// Mitsubishi GX Works2 project: 412_Coating_Code   PLC: Q03UDE

PROGRAM MAIN
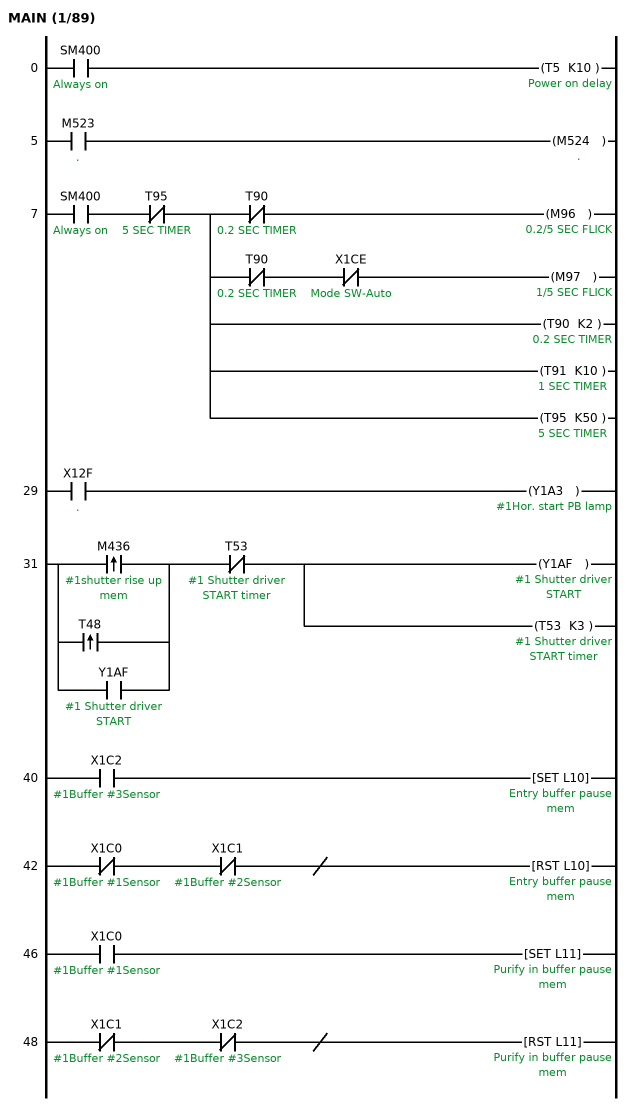
0     LD      SM400  ; Always on
      OUT     T5 K10  ; Power on delay
5     LD      M523  ; .
      OUT     M524  ; .
7     LD      SM400  ; Always on
      ANI     T95  ; 5 SEC TIMER
      MPS
      ANI     T90  ; 0.2 SEC TIMER
      OUT     M96  ; 0.2/5 SEC FLICK
      MRD
      ANI     T90  ; 0.2 SEC TIMER
      ANI     X1CE  ; Mode SW-Auto
      OUT     M97  ; 1/5 SEC FLICK
      MPP
      OUT     T90 K2  ; 0.2 SEC TIMER
      OUT     T91 K10  ; 1 SEC TIMER
      OUT     T95 K50  ; 5 SEC TIMER
29    LD      X12F  ; .
      OUT     Y1A3  ; #1Hor. start PB lamp
31    LDP     M436  ; #1shutter rise up mem
      ORP     T48
      OR      Y1AF  ; #1 Shutter driver START
      ANI     T53  ; #1 Shutter driver START timer
      OUT     Y1AF  ; #1 Shutter driver START
      OUT     T53 K3  ; #1 Shutter driver START timer
40    LD      X1C2  ; #1Buffer #3Sensor
      SET     L10  ; Entry buffer pause mem
42    LDI     X1C0  ; #1Buffer #1Sensor
      ANI     X1C1  ; #1Buffer #2Sensor
      INV
      RST     L10  ; Entry buffer pause mem
46    LD      X1C0  ; #1Buffer #1Sensor
      SET     L11  ; Purify in buffer pause mem
48    LDI     X1C1  ; #1Buffer #2Sensor
      ANI     X1C2  ; #1Buffer #3Sensor
      INV
      RST     L11  ; Purify in buffer pause mem
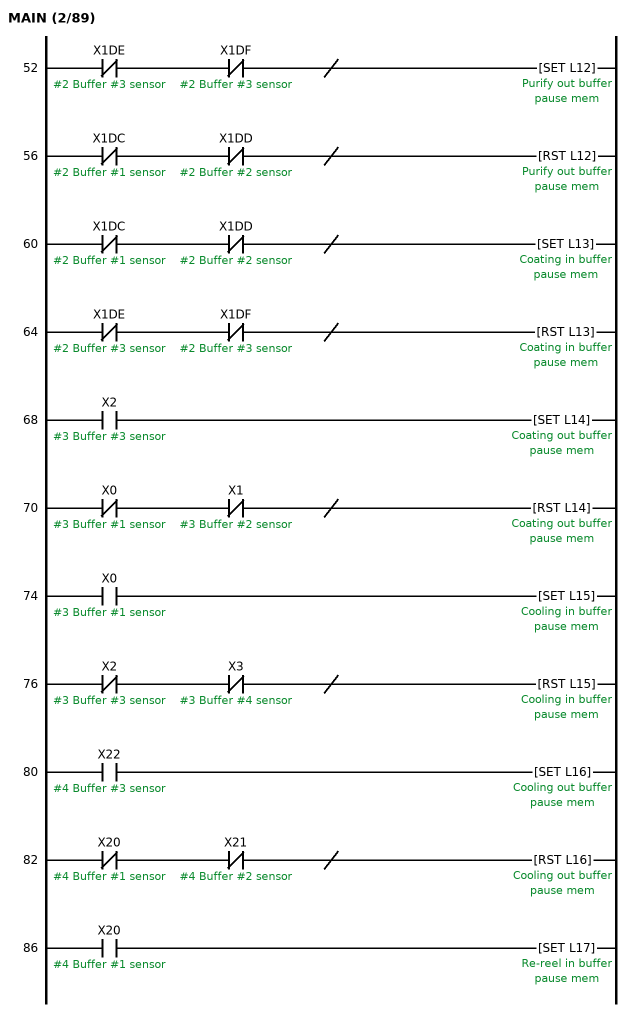
52    LDI     X1DE  ; #2 Buffer #3 sensor
      ANI     X1DF  ; #2 Buffer #3 sensor
      INV
      SET     L12  ; Purify out buffer pause mem
56    LDI     X1DC  ; #2 Buffer #1 sensor
      ANI     X1DD  ; #2 Buffer #2 sensor
      INV
      RST     L12  ; Purify out buffer pause mem
60    LDI     X1DC  ; #2 Buffer #1 sensor
      ANI     X1DD  ; #2 Buffer #2 sensor
      INV
      SET     L13  ; Coating in buffer pause mem
64    LDI     X1DE  ; #2 Buffer #3 sensor
      ANI     X1DF  ; #2 Buffer #3 sensor
      INV
      RST     L13  ; Coating in buffer pause mem
68    LD      X2  ; #3 Buffer #3 sensor
      SET     L14  ; Coating out buffer pause mem
70    LDI     X0  ; #3 Buffer #1 sensor
      ANI     X1  ; #3 Buffer #2 sensor
      INV
      RST     L14  ; Coating out buffer pause mem
74    LD      X0  ; #3 Buffer #1 sensor
      SET     L15  ; Cooling in buffer pause mem
76    LDI     X2  ; #3 Buffer #3 sensor
      ANI     X3  ; #3 Buffer #4 sensor
      INV
      RST     L15  ; Cooling in buffer pause mem
80    LD      X22  ; #4 Buffer #3 sensor
      SET     L16  ; Cooling out buffer pause mem
82    LDI     X20  ; #4 Buffer #1 sensor
      ANI     X21  ; #4 Buffer #2 sensor
      INV
      RST     L16  ; Cooling out buffer pause mem
86    LD      X20  ; #4 Buffer #1 sensor
      SET     L17  ; Re-reel in buffer pause mem
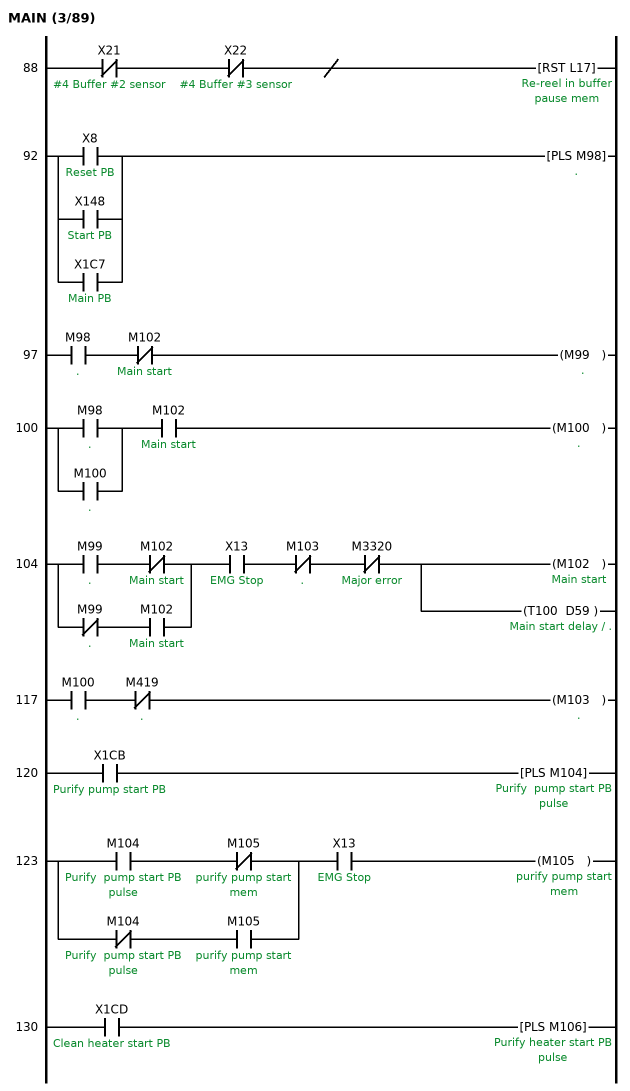
88    LDI     X21  ; #4 Buffer #2 sensor
      ANI     X22  ; #4 Buffer #3 sensor
      INV
      RST     L17  ; Re-reel in buffer pause mem
92    LD      X8  ; Reset PB
      OR      X148  ; Start PB
      OR      X1C7  ; Main PB
      PLS     M98  ; .
97    LD      M98  ; .
      ANI     M102  ; Main start
      OUT     M99  ; .
100   LD      M98  ; .
      OR      M100  ; .
      AND     M102  ; Main start
      OUT     M100  ; .
104   LD      M99  ; .
      ANI     M102  ; Main start
      LDI     M99  ; .
      AND     M102  ; Main start
      ORB
      AND     X13  ; EMG Stop
      ANI     M103  ; .
      ANI     M3320  ; Major error
      OUT     M102  ; Main start
      OUT     T100 D59  ; Main start delay / .
117   LD      M100  ; .
      ANI     M419  ; .
      OUT     M103  ; .
120   LD      X1CB  ; Purify pump start PB
      PLS     M104  ; Purify  pump start PB pulse
123   LD      M104  ; Purify  pump start PB pulse
      ANI     M105  ; purify pump start mem
      LDI     M104  ; Purify  pump start PB pulse
      AND     M105  ; purify pump start mem
      ORB
      AND     X13  ; EMG Stop
      OUT     M105  ; purify pump start mem
130   LD      X1CD  ; Clean heater start PB
      PLS     M106  ; Purify heater start PB pulse
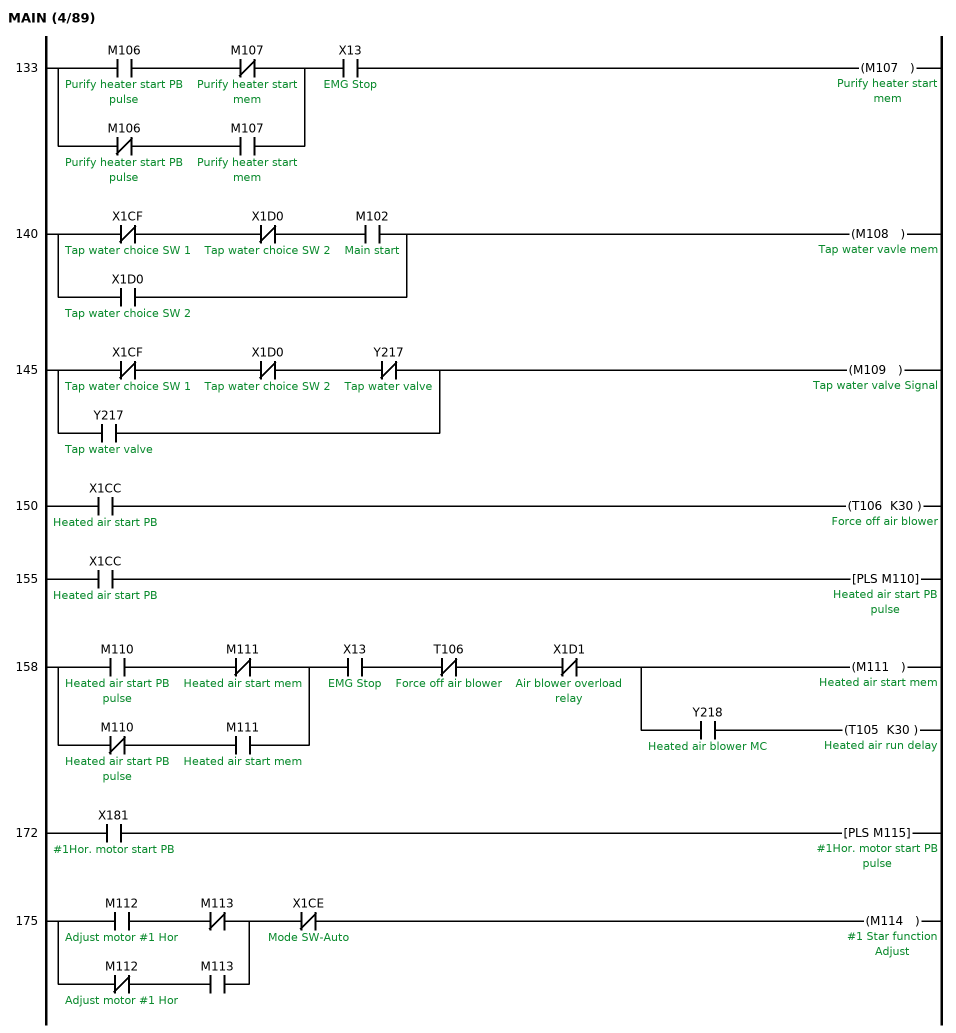
133   LD      M106  ; Purify heater start PB pulse
      ANI     M107  ; Purify heater start mem
      LDI     M106  ; Purify heater start PB pulse
      AND     M107  ; Purify heater start mem
      ORB
      AND     X13  ; EMG Stop
      OUT     M107  ; Purify heater start mem
140   LDI     X1CF  ; Tap water choice SW 1
      ANI     X1D0  ; Tap water choice SW 2
      AND     M102  ; Main start
      OR      X1D0  ; Tap water choice SW 2
      OUT     M108  ; Tap water vavle mem
145   LDI     X1CF  ; Tap water choice SW 1
      ANI     X1D0  ; Tap water choice SW 2
      ANI     Y217  ; Tap water valve
      OR      Y217  ; Tap water valve
      OUT     M109  ; Tap water valve Signal
150   LD      X1CC  ; Heated air start PB
      OUT     T106 K30  ; Force off air blower
155   LD      X1CC  ; Heated air start PB
      PLS     M110  ; Heated air start PB pulse
158   LD      M110  ; Heated air start PB pulse
      ANI     M111  ; Heated air start mem
      LDI     M110  ; Heated air start PB pulse
      AND     M111  ; Heated air start mem
      ORB
      AND     X13  ; EMG Stop
      ANI     T106  ; Force off air blower
      ANI     X1D1  ; Air blower overload relay
      OUT     M111  ; Heated air start mem
      AND     Y218  ; Heated air blower MC
      OUT     T105 K30  ; Heated air run delay
172   LD      X181  ; #1Hor. motor start PB
      PLS     M115  ; #1Hor. motor start PB pulse
175   LD      M112  ; Adjust motor #1 Hor
      ANI     M113
      LDI     M112  ; Adjust motor #1 Hor
      AND     M113
      ORB
      ANI     X1CE  ; Mode SW-Auto
      OUT     M114  ; #1 Star function Adjust
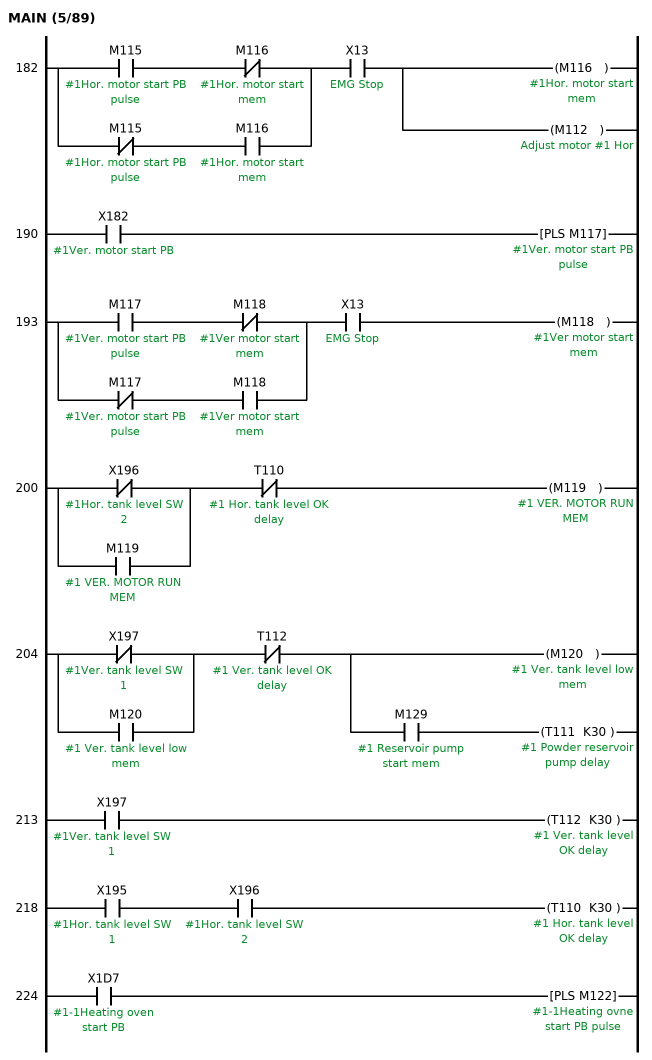
182   LD      M115  ; #1Hor. motor start PB pulse
      ANI     M116  ; #1Hor. motor start mem
      LDI     M115  ; #1Hor. motor start PB pulse
      AND     M116  ; #1Hor. motor start mem
      ORB
      AND     X13  ; EMG Stop
      OUT     M116  ; #1Hor. motor start mem
      OUT     M112  ; Adjust motor #1 Hor
190   LD      X182  ; #1Ver. motor start PB
      PLS     M117  ; #1Ver. motor start PB pulse
193   LD      M117  ; #1Ver. motor start PB pulse
      ANI     M118  ; #1Ver motor start mem
      LDI     M117  ; #1Ver. motor start PB pulse
      AND     M118  ; #1Ver motor start mem
      ORB
      AND     X13  ; EMG Stop
      OUT     M118  ; #1Ver motor start mem
200   LDI     X196  ; #1Hor. tank level SW 2
      OR      M119  ; #1 VER. MOTOR RUN MEM
      ANI     T110  ; #1 Hor. tank level OK delay
      OUT     M119  ; #1 VER. MOTOR RUN MEM
204   LDI     X197  ; #1Ver. tank level SW 1
      OR      M120  ; #1 Ver. tank level low mem
      ANI     T112  ; #1 Ver. tank level OK delay
      OUT     M120  ; #1 Ver. tank level low mem
      AND     M129  ; #1 Reservoir pump start mem
      OUT     T111 K30  ; #1 Powder reservoir pump delay
213   LD      X197  ; #1Ver. tank level SW 1
      OUT     T112 K30  ; #1 Ver. tank level OK delay
218   LD      X195  ; #1Hor. tank level SW 1
      AND     X196  ; #1Hor. tank level SW 2
      OUT     T110 K30  ; #1 Hor. tank level OK delay
224   LD      X1D7  ; #1-1Heating oven start PB
      PLS     M122  ; #1-1Heating ovne start PB pulse
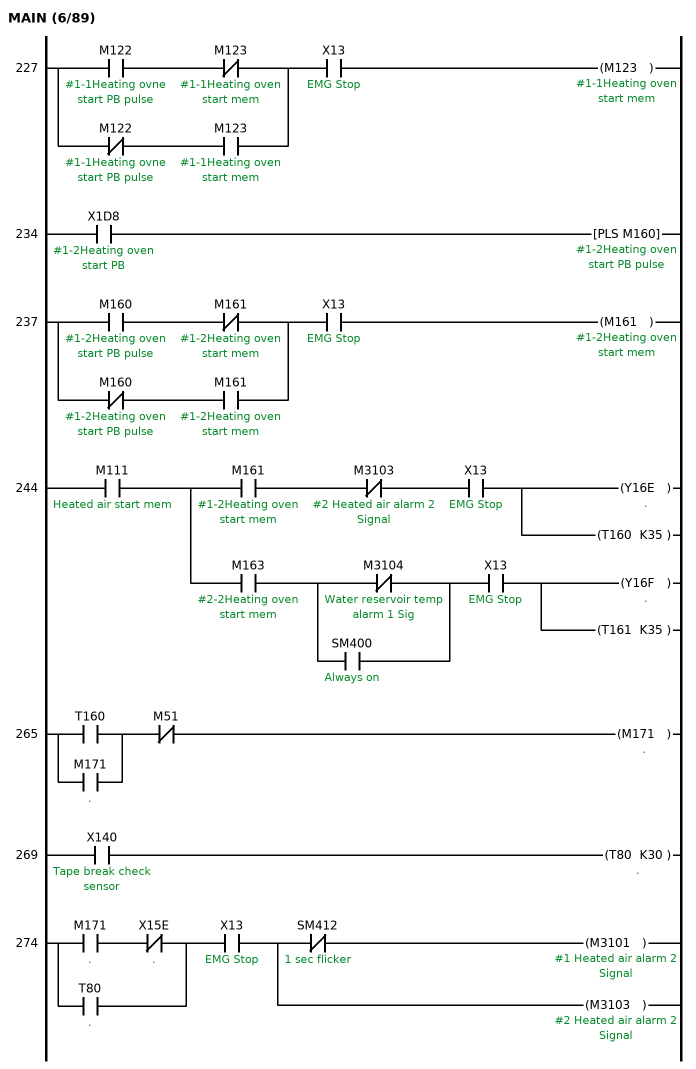
227   LD      M122  ; #1-1Heating ovne start PB pulse
      ANI     M123  ; #1-1Heating oven start mem
      LDI     M122  ; #1-1Heating ovne start PB pulse
      AND     M123  ; #1-1Heating oven start mem
      ORB
      AND     X13  ; EMG Stop
      OUT     M123  ; #1-1Heating oven start mem
234   LD      X1D8  ; #1-2Heating oven start PB
      PLS     M160  ; #1-2Heating oven start PB pulse
237   LD      M160  ; #1-2Heating oven start PB pulse
      ANI     M161  ; #1-2Heating oven start mem
      LDI     M160  ; #1-2Heating oven start PB pulse
      AND     M161  ; #1-2Heating oven start mem
      ORB
      AND     X13  ; EMG Stop
      OUT     M161  ; #1-2Heating oven start mem
244   LD      M111  ; Heated air start mem
      MPS
      AND     M161  ; #1-2Heating oven start mem
      ANI     M3103  ; #2 Heated air alarm 2 Signal
      AND     X13  ; EMG Stop
      OUT     Y16E  ; .
      OUT     T160 K35
      MPP
      AND     M163  ; #2-2Heating oven start mem
      LDI     M3104  ; Water reservoir temp alarm 1 Sig
      OR      SM400  ; Always on
      ANB
      AND     X13  ; EMG Stop
      OUT     Y16F  ; .
      OUT     T161 K35
265   LD      T160
      OR      M171  ; .
      ANI     M51
      OUT     M171  ; .
269   LD      X140  ; Tape break check sensor
      OUT     T80 K30  ; .
274   LD      M171  ; .
      ANI     X15E  ; .
      OR      T80  ; .
      AND     X13  ; EMG Stop
      MPS
      ANI     SM412  ; 1 sec flicker
      OUT     M3101  ; #1 Heated air alarm 2 Signal
      MPP
      OUT     M3103  ; #2 Heated air alarm 2 Signal
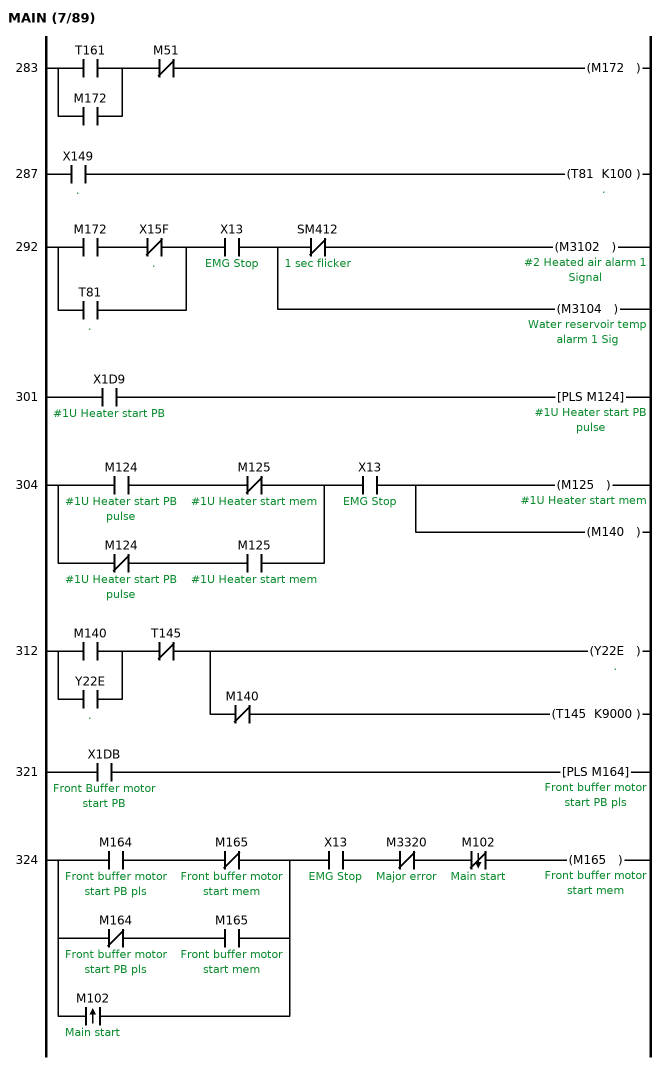
283   LD      T161
      OR      M172
      ANI     M51
      OUT     M172
287   LD      X149  ; .
      OUT     T81 K100  ; .
292   LD      M172
      ANI     X15F  ; .
      OR      T81  ; .
      AND     X13  ; EMG Stop
      MPS
      ANI     SM412  ; 1 sec flicker
      OUT     M3102  ; #2 Heated air alarm 1 Signal
      MPP
      OUT     M3104  ; Water reservoir temp alarm 1 Sig
301   LD      X1D9  ; #1U Heater start PB
      PLS     M124  ; #1U Heater start PB pulse
304   LD      M124  ; #1U Heater start PB pulse
      ANI     M125  ; #1U Heater start mem
      LDI     M124  ; #1U Heater start PB pulse
      AND     M125  ; #1U Heater start mem
      ORB
      AND     X13  ; EMG Stop
      OUT     M125  ; #1U Heater start mem
      OUT     M140
312   LD      M140
      OR      Y22E  ; .
      ANI     T145
      OUT     Y22E  ; .
      ANI     M140
      OUT     T145 K9000
321   LD      X1DB  ; Front Buffer motor start PB
      PLS     M164  ; Front buffer motor start PB pls
324   LD      M164  ; Front buffer motor start PB pls
      ANI     M165  ; Front buffer motor start mem
      LDI     M164  ; Front buffer motor start PB pls
      AND     M165  ; Front buffer motor start mem
      ORB
      ORP     M102  ; Main start
      AND     X13  ; EMG Stop
      ANI     M3320  ; Major error
      ANDFI   M102  ; Main start
      OUT     M165  ; Front buffer motor start mem
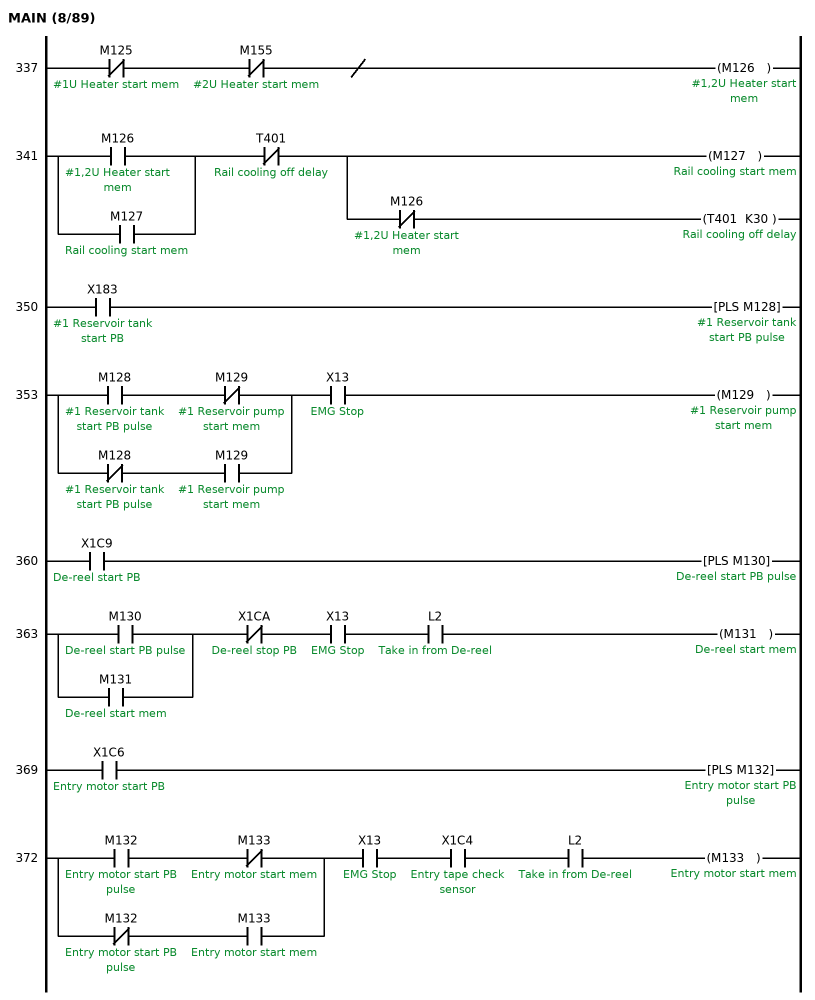
337   LDI     M125  ; #1U Heater start mem
      ANI     M155  ; #2U Heater start mem
      INV
      OUT     M126  ; #1,2U Heater start mem
341   LD      M126  ; #1,2U Heater start mem
      OR      M127  ; Rail cooling start mem
      ANI     T401  ; Rail cooling off delay
      OUT     M127  ; Rail cooling start mem
      ANI     M126  ; #1,2U Heater start mem
      OUT     T401 K30  ; Rail cooling off delay
350   LD      X183  ; #1 Reservoir tank start PB
      PLS     M128  ; #1 Reservoir tank start PB pulse
353   LD      M128  ; #1 Reservoir tank start PB pulse
      ANI     M129  ; #1 Reservoir pump start mem
      LDI     M128  ; #1 Reservoir tank start PB pulse
      AND     M129  ; #1 Reservoir pump start mem
      ORB
      AND     X13  ; EMG Stop
      OUT     M129  ; #1 Reservoir pump start mem
360   LD      X1C9  ; De-reel start PB
      PLS     M130  ; De-reel start PB pulse
363   LD      M130  ; De-reel start PB pulse
      OR      M131  ; De-reel start mem
      ANI     X1CA  ; De-reel stop PB
      AND     X13  ; EMG Stop
      AND     L2  ; Take in from De-reel
      OUT     M131  ; De-reel start mem
369   LD      X1C6  ; Entry motor start PB
      PLS     M132  ; Entry motor start PB pulse
372   LD      M132  ; Entry motor start PB pulse
      ANI     M133  ; Entry motor start mem
      LDI     M132  ; Entry motor start PB pulse
      AND     M133  ; Entry motor start mem
      ORB
      AND     X13  ; EMG Stop
      AND     X1C4  ; Entry tape check sensor
      AND     L2  ; Take in from De-reel
      OUT     M133  ; Entry motor start mem
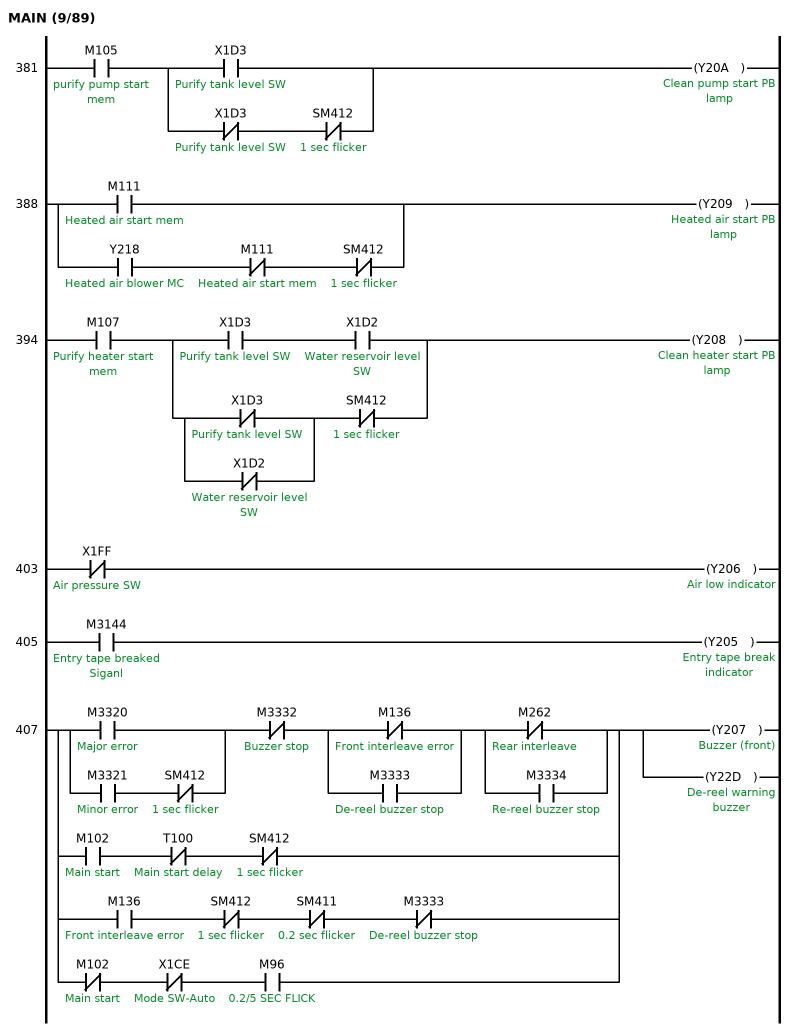
381   LD      M105  ; purify pump start mem
      LD      X1D3  ; Purify tank level SW
      LDI     X1D3  ; Purify tank level SW
      ANI     SM412  ; 1 sec flicker
      ORB
      ANB
      OUT     Y20A  ; Clean pump start PB lamp
388   LD      M111  ; Heated air start mem
      LD      Y218  ; Heated air blower MC
      ANI     M111  ; Heated air start mem
      ANI     SM412  ; 1 sec flicker
      ORB
      OUT     Y209  ; Heated air start PB lamp
394   LD      M107  ; Purify heater start mem
      LD      X1D3  ; Purify tank level SW
      AND     X1D2  ; Water reservoir level SW
      LDI     X1D3  ; Purify tank level SW
      ORI     X1D2  ; Water reservoir level SW
      ANI     SM412  ; 1 sec flicker
      ORB
      ANB
      OUT     Y208  ; Clean heater start PB lamp
403   LDI     X1FF  ; Air pressure SW
      OUT     Y206  ; Air low indicator
405   LD      M3144  ; Entry tape breaked Siganl
      OUT     Y205  ; Entry tape break indicator
407   LD      M3320  ; Major error
      LD      M3321  ; Minor error
      ANI     SM412  ; 1 sec flicker
      ORB
      ANI     M3332  ; Buzzer stop
      LDI     M136  ; Front interleave error
      OR      M3333  ; De-reel buzzer stop
      ANB
      LDI     M262  ; Rear interleave
      OR      M3334  ; Re-reel buzzer stop
      ANB
      LD      M102  ; Main start
      ANI     T100  ; Main start delay
      ANI     SM412  ; 1 sec flicker
      ORB
      LD      M136  ; Front interleave error
      ANI     SM412  ; 1 sec flicker
      ANI     SM411  ; 0.2 sec flicker
      ANI     M3333  ; De-reel buzzer stop
      ORB
      LDI     M102  ; Main start
      ANI     X1CE  ; Mode SW-Auto
      AND     M96  ; 0.2/5 SEC FLICK
      ORB
      OUT     Y207  ; Buzzer (front)
      OUT     Y22D  ; De-reel warning buzzer
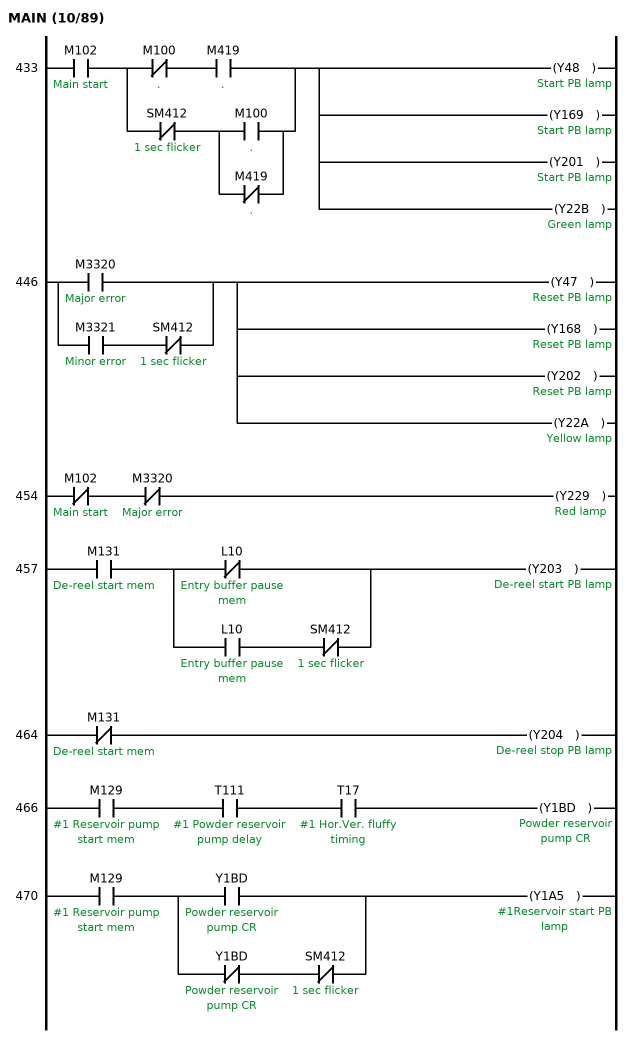
433   LD      M102  ; Main start
      LDI     M100  ; .
      AND     M419  ; .
      LDI     SM412  ; 1 sec flicker
      LD      M100  ; .
      ORI     M419  ; .
      ANB
      ORB
      ANB
      OUT     Y48  ; Start PB lamp
      OUT     Y169  ; Start PB lamp
      OUT     Y201  ; Start PB lamp
      OUT     Y22B  ; Green lamp
446   LD      M3320  ; Major error
      LD      M3321  ; Minor error
      ANI     SM412  ; 1 sec flicker
      ORB
      OUT     Y47  ; Reset PB lamp
      OUT     Y168  ; Reset PB lamp
      OUT     Y202  ; Reset PB lamp
      OUT     Y22A  ; Yellow lamp
454   LDI     M102  ; Main start
      ANI     M3320  ; Major error
      OUT     Y229  ; Red lamp
457   LD      M131  ; De-reel start mem
      LDI     L10  ; Entry buffer pause mem
      LD      L10  ; Entry buffer pause mem
      ANI     SM412  ; 1 sec flicker
      ORB
      ANB
      OUT     Y203  ; De-reel start PB lamp
464   LDI     M131  ; De-reel start mem
      OUT     Y204  ; De-reel stop PB lamp
466   LD      M129  ; #1 Reservoir pump start mem
      AND     T111  ; #1 Powder reservoir pump delay
      AND     T17  ; #1 Hor.Ver. fluffy timing
      OUT     Y1BD  ; Powder reservoir pump CR
470   LD      M129  ; #1 Reservoir pump start mem
      LD      Y1BD  ; Powder reservoir pump CR
      LDI     Y1BD  ; Powder reservoir pump CR
      ANI     SM412  ; 1 sec flicker
      ORB
      ANB
      OUT     Y1A5  ; #1Reservoir start PB lamp
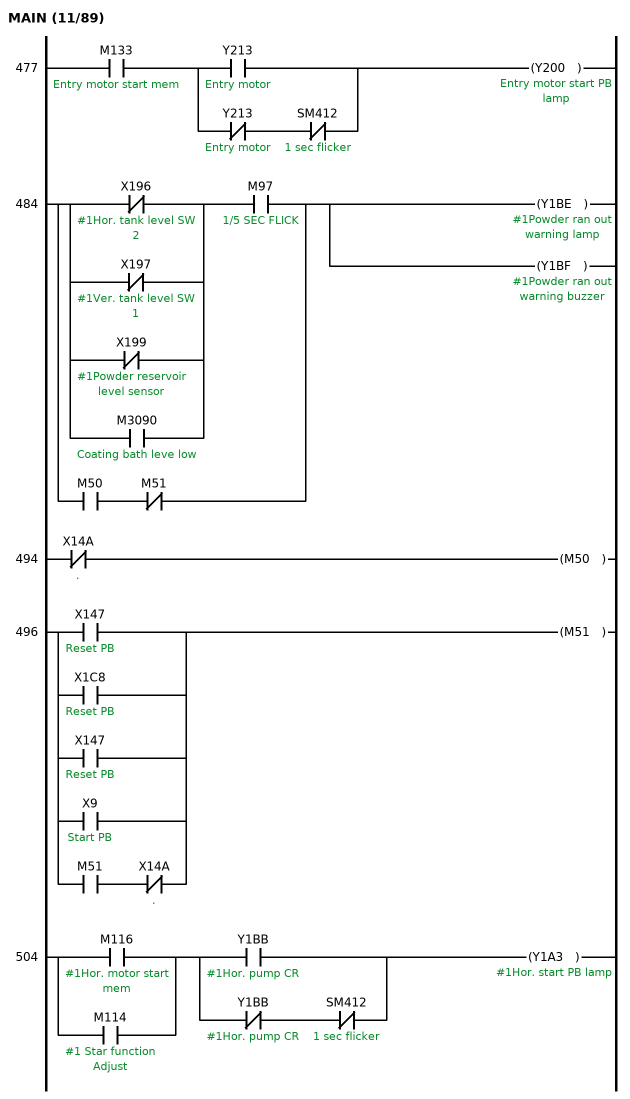
477   LD      M133  ; Entry motor start mem
      LD      Y213  ; Entry motor
      LDI     Y213  ; Entry motor
      ANI     SM412  ; 1 sec flicker
      ORB
      ANB
      OUT     Y200  ; Entry motor start PB lamp
484   LDI     X196  ; #1Hor. tank level SW 2
      ORI     X197  ; #1Ver. tank level SW 1
      ORI     X199  ; #1Powder reservoir level sensor
      OR      M3090  ; Coating bath leve low
      AND     M97  ; 1/5 SEC FLICK
      LD      M50
      ANI     M51
      ORB
      OUT     Y1BE  ; #1Powder ran out warning lamp
      OUT     Y1BF  ; #1Powder ran out warning buzzer
494   LDI     X14A  ; .
      OUT     M50
496   LD      X147  ; Reset PB
      OR      X1C8  ; Reset PB
      OR      X147  ; Reset PB
      OR      X9  ; Start PB
      LD      M51
      ANI     X14A  ; .
      ORB
      OUT     M51
504   LD      M116  ; #1Hor. motor start mem
      OR      M114  ; #1 Star function Adjust
      LD      Y1BB  ; #1Hor. pump CR
      LDI     Y1BB  ; #1Hor. pump CR
      ANI     SM412  ; 1 sec flicker
      ORB
      ANB
      OUT     Y1A3  ; #1Hor. start PB lamp
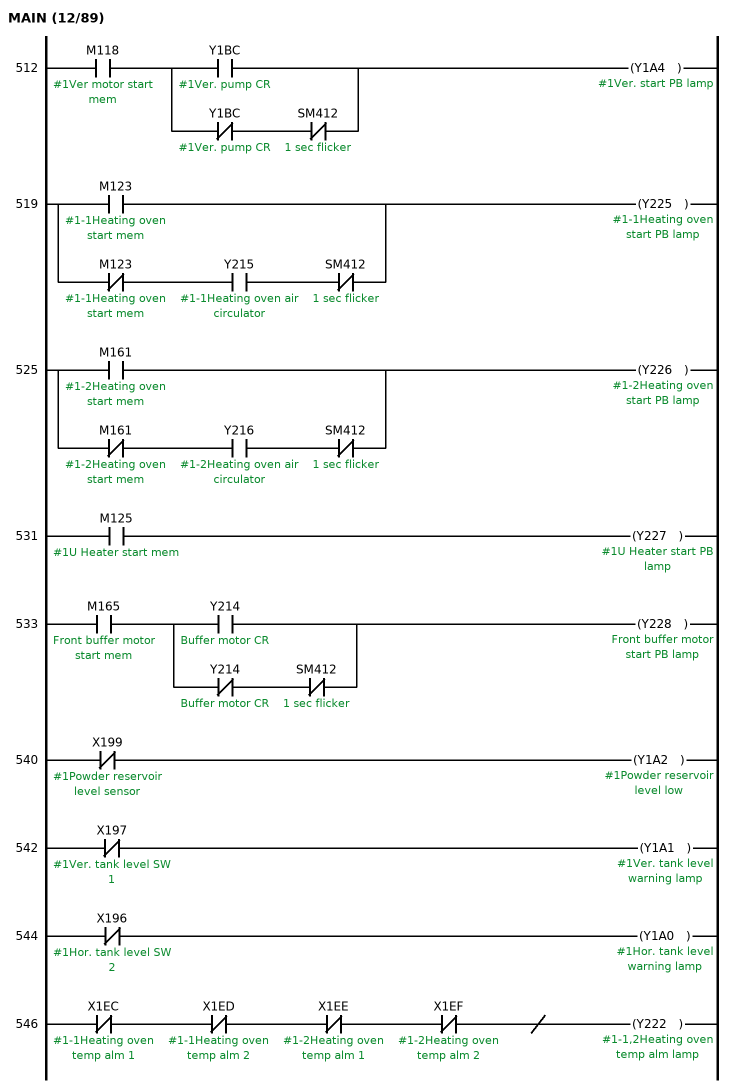
512   LD      M118  ; #1Ver motor start mem
      LD      Y1BC  ; #1Ver. pump CR
      LDI     Y1BC  ; #1Ver. pump CR
      ANI     SM412  ; 1 sec flicker
      ORB
      ANB
      OUT     Y1A4  ; #1Ver. start PB lamp
519   LD      M123  ; #1-1Heating oven start mem
      LDI     M123  ; #1-1Heating oven start mem
      AND     Y215  ; #1-1Heating oven air circulator
      ANI     SM412  ; 1 sec flicker
      ORB
      OUT     Y225  ; #1-1Heating oven start PB lamp
525   LD      M161  ; #1-2Heating oven start mem
      LDI     M161  ; #1-2Heating oven start mem
      AND     Y216  ; #1-2Heating oven air circulator
      ANI     SM412  ; 1 sec flicker
      ORB
      OUT     Y226  ; #1-2Heating oven start PB lamp
531   LD      M125  ; #1U Heater start mem
      OUT     Y227  ; #1U Heater start PB lamp
533   LD      M165  ; Front buffer motor start mem
      LD      Y214  ; Buffer motor CR
      LDI     Y214  ; Buffer motor CR
      ANI     SM412  ; 1 sec flicker
      ORB
      ANB
      OUT     Y228  ; Front buffer motor start PB lamp
540   LDI     X199  ; #1Powder reservoir level sensor
      OUT     Y1A2  ; #1Powder reservoir level low
542   LDI     X197  ; #1Ver. tank level SW 1
      OUT     Y1A1  ; #1Ver. tank level warning lamp
544   LDI     X196  ; #1Hor. tank level SW 2
      OUT     Y1A0  ; #1Hor. tank level warning lamp
546   LDI     X1EC  ; #1-1Heating oven temp alm 1
      ANI     X1ED  ; #1-1Heating oven temp alm 2
      ANI     X1EE  ; #1-2Heating oven temp alm 1
      ANI     X1EF  ; #1-2Heating oven temp alm 2
      INV
      OUT     Y222  ; #1-1,2Heating oven temp alm lamp
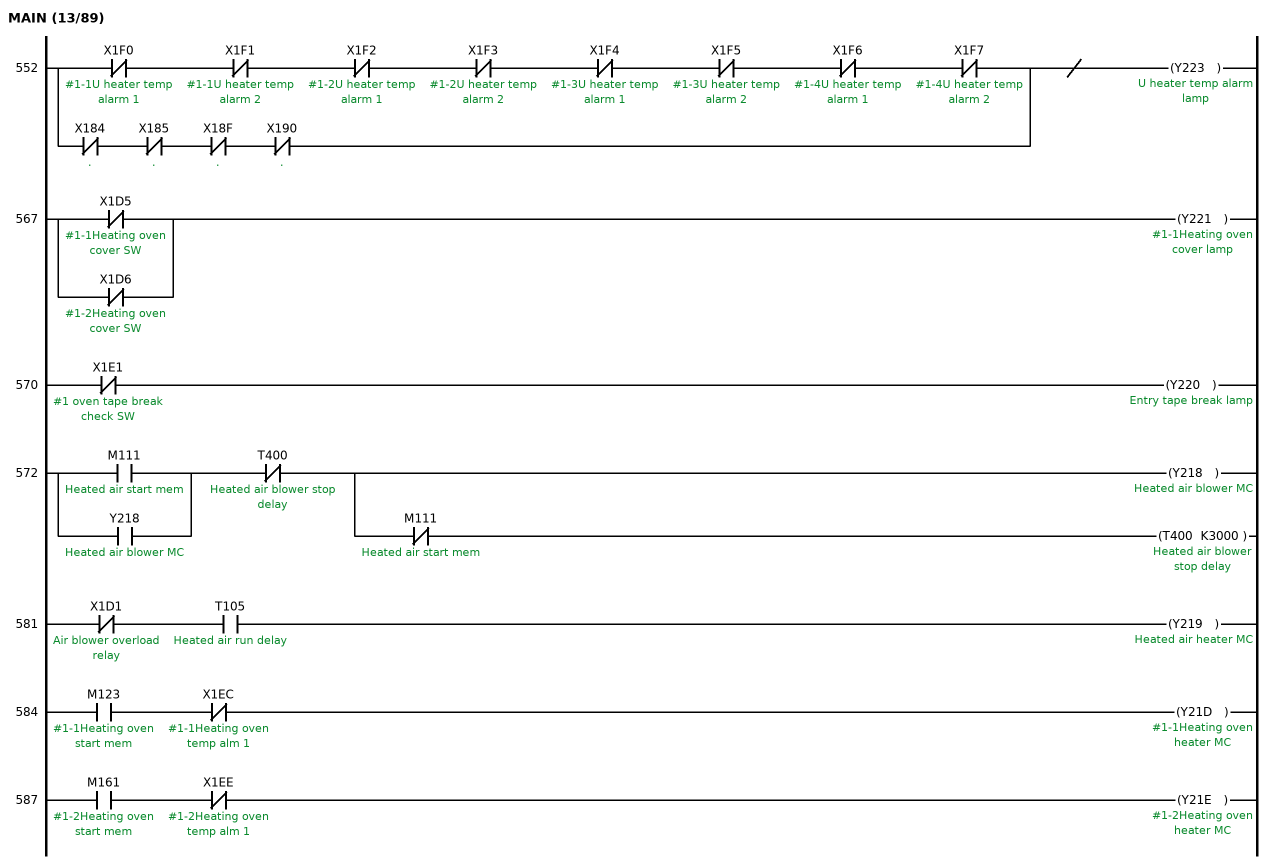
552   LDI     X1F0  ; #1-1U heater temp alarm 1
      ANI     X1F1  ; #1-1U heater temp alarm 2
      ANI     X1F2  ; #1-2U heater temp alarm 1
      ANI     X1F3  ; #1-2U heater temp alarm 2
      ANI     X1F4  ; #1-3U heater temp alarm 1
      ANI     X1F5  ; #1-3U heater temp alarm 2
      ANI     X1F6  ; #1-4U heater temp alarm 1
      ANI     X1F7  ; #1-4U heater temp alarm 2
      LDI     X184  ; .
      ANI     X185  ; .
      ANI     X18F  ; .
      ANI     X190  ; .
      ORB
      INV
      OUT     Y223  ; U heater temp alarm lamp
567   LDI     X1D5  ; #1-1Heating oven cover SW
      ORI     X1D6  ; #1-2Heating oven cover SW
      OUT     Y221  ; #1-1Heating oven cover lamp
570   LDI     X1E1  ; #1 oven tape break check SW
      OUT     Y220  ; Entry tape break lamp
572   LD      M111  ; Heated air start mem
      OR      Y218  ; Heated air blower MC
      ANI     T400  ; Heated air blower stop delay
      OUT     Y218  ; Heated air blower MC
      ANI     M111  ; Heated air start mem
      OUT     T400 K3000  ; Heated air blower stop delay
581   LDI     X1D1  ; Air blower overload relay
      AND     T105  ; Heated air run delay
      OUT     Y219  ; Heated air heater MC
584   LD      M123  ; #1-1Heating oven start mem
      ANI     X1EC  ; #1-1Heating oven temp alm 1
      OUT     Y21D  ; #1-1Heating oven heater MC
587   LD      M161  ; #1-2Heating oven start mem
      ANI     X1EE  ; #1-2Heating oven temp alm 1
      OUT     Y21E  ; #1-2Heating oven heater MC
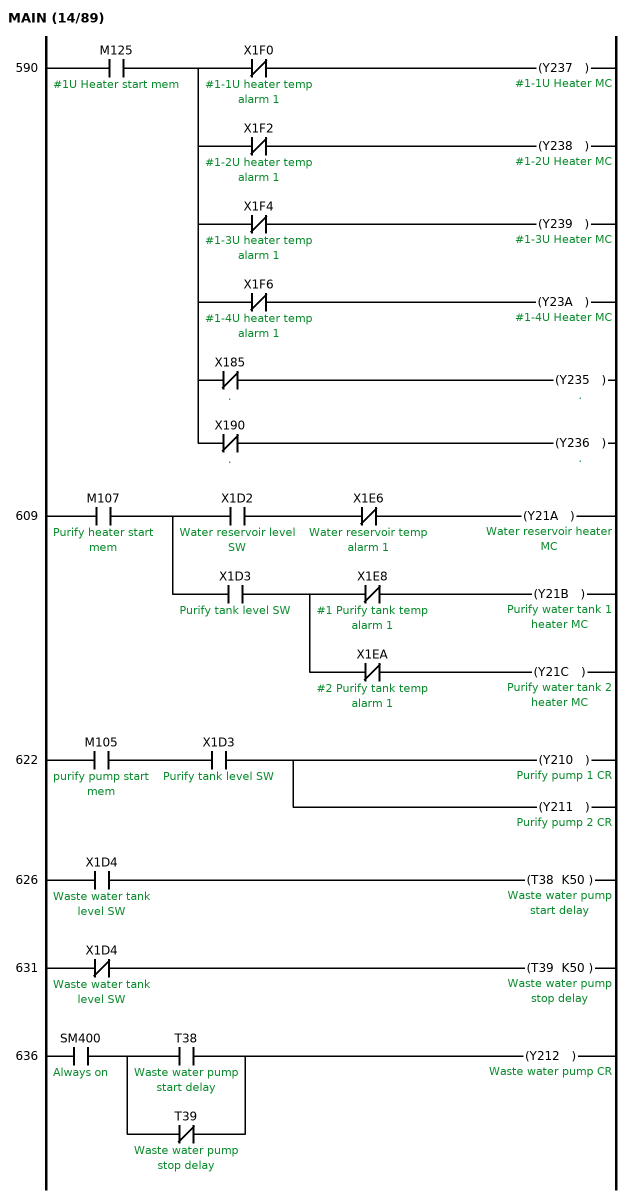
590   LD      M125  ; #1U Heater start mem
      MPS
      ANI     X1F0  ; #1-1U heater temp alarm 1
      OUT     Y237  ; #1-1U Heater MC
      MRD
      ANI     X1F2  ; #1-2U heater temp alarm 1
      OUT     Y238  ; #1-2U Heater MC
      MRD
      ANI     X1F4  ; #1-3U heater temp alarm 1
      OUT     Y239  ; #1-3U Heater MC
      MRD
      ANI     X1F6  ; #1-4U heater temp alarm 1
      OUT     Y23A  ; #1-4U Heater MC
      MRD
      ANI     X185  ; .
      OUT     Y235  ; .
      MPP
      ANI     X190  ; .
      OUT     Y236  ; .
609   LD      M107  ; Purify heater start mem
      MPS
      AND     X1D2  ; Water reservoir level SW
      ANI     X1E6  ; Water reservoir temp alarm 1
      OUT     Y21A  ; Water reservoir heater MC
      MPP
      AND     X1D3  ; Purify tank level SW
      MPS
      ANI     X1E8  ; #1 Purify tank temp alarm 1
      OUT     Y21B  ; Purify water tank 1 heater MC
      MPP
      ANI     X1EA  ; #2 Purify tank temp alarm 1
      OUT     Y21C  ; Purify water tank 2 heater MC
622   LD      M105  ; purify pump start mem
      AND     X1D3  ; Purify tank level SW
      OUT     Y210  ; Purify pump 1 CR
      OUT     Y211  ; Purify pump 2 CR
626   LD      X1D4  ; Waste water tank level SW
      OUT     T38 K50  ; Waste water pump start delay
631   LDI     X1D4  ; Waste water tank level SW
      OUT     T39 K50  ; Waste water pump stop delay
636   LD      SM400  ; Always on
      LD      T38  ; Waste water pump start delay
      ORI     T39  ; Waste water pump stop delay
      ANB
      OUT     Y212  ; Waste water pump CR
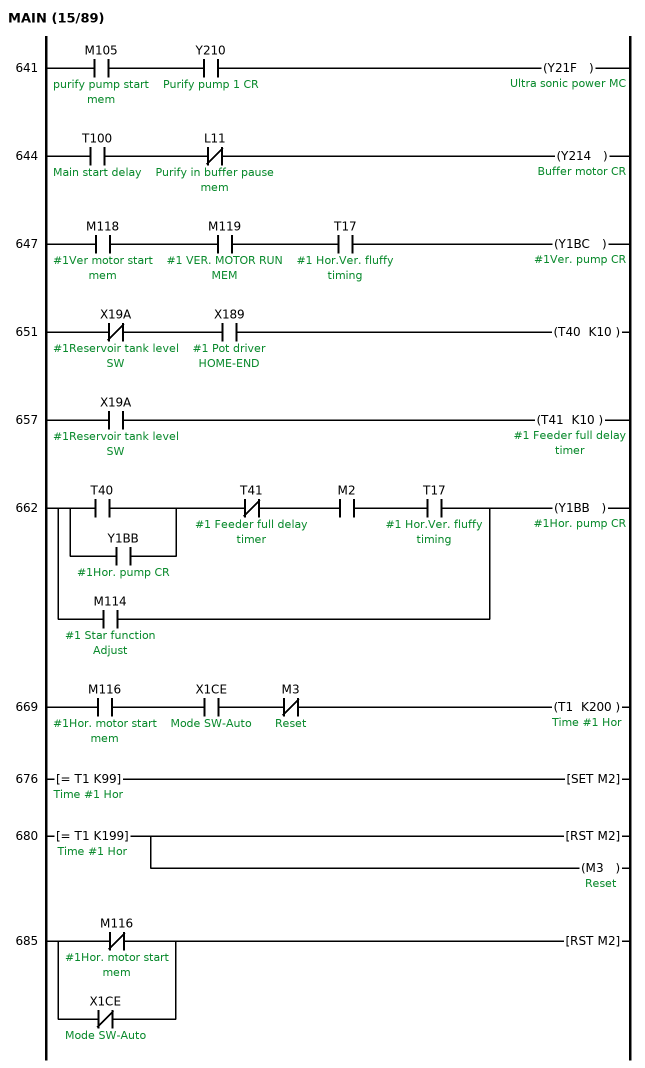
641   LD      M105  ; purify pump start mem
      AND     Y210  ; Purify pump 1 CR
      OUT     Y21F  ; Ultra sonic power MC
644   LD      T100  ; Main start delay
      ANI     L11  ; Purify in buffer pause mem
      OUT     Y214  ; Buffer motor CR
647   LD      M118  ; #1Ver motor start mem
      AND     M119  ; #1 VER. MOTOR RUN MEM
      AND     T17  ; #1 Hor.Ver. fluffy timing
      OUT     Y1BC  ; #1Ver. pump CR
651   LDI     X19A  ; #1Reservoir tank level SW
      AND     X189  ; #1 Pot driver HOME-END
      OUT     T40 K10
657   LD      X19A  ; #1Reservoir tank level SW
      OUT     T41 K10  ; #1 Feeder full delay timer
662   LD      T40
      OR      Y1BB  ; #1Hor. pump CR
      ANI     T41  ; #1 Feeder full delay timer
      AND     M2
      AND     T17  ; #1 Hor.Ver. fluffy timing
      OR      M114  ; #1 Star function Adjust
      OUT     Y1BB  ; #1Hor. pump CR
669   LD      M116  ; #1Hor. motor start mem
      AND     X1CE  ; Mode SW-Auto
      ANI     M3  ; Reset
      OUT     T1 K200  ; Time #1 Hor
676   LD=     T1 K99  ; Time #1 Hor
      SET     M2
680   LD=     T1 K199  ; Time #1 Hor
      RST     M2
      OUT     M3  ; Reset
685   LDI     M116  ; #1Hor. motor start mem
      ORI     X1CE  ; Mode SW-Auto
      RST     M2
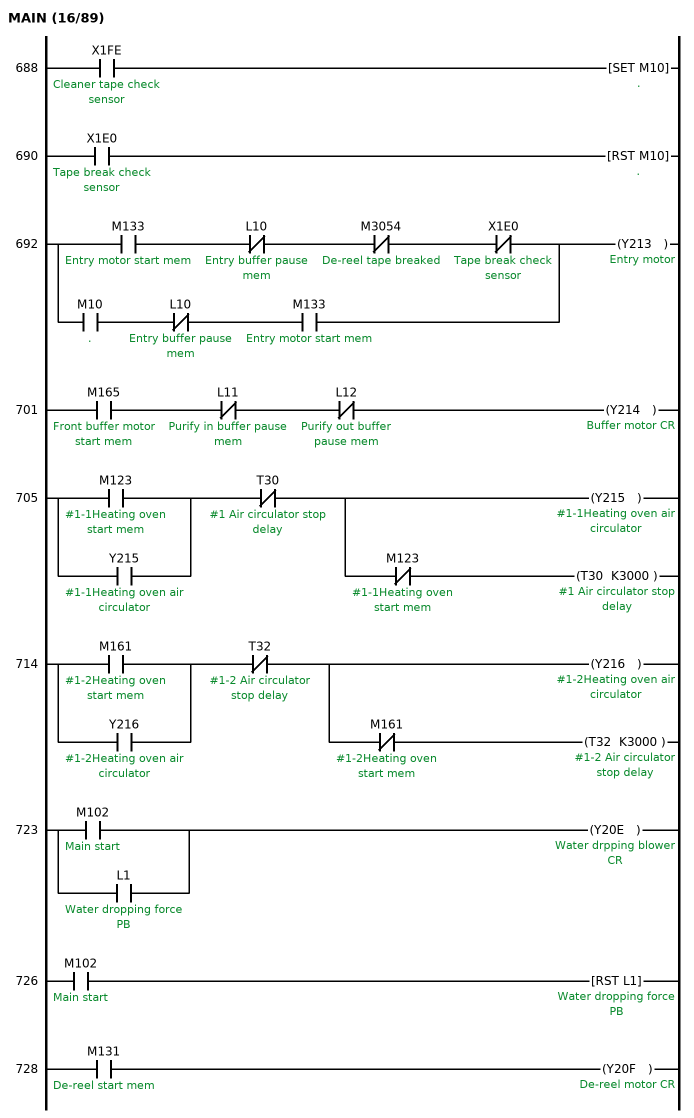
688   LD      X1FE  ; Cleaner tape check sensor
      SET     M10  ; .
690   LD      X1E0  ; Tape break check sensor
      RST     M10  ; .
692   LD      M133  ; Entry motor start mem
      ANI     L10  ; Entry buffer pause mem
      ANI     M3054  ; De-reel tape breaked
      ANI     X1E0  ; Tape break check sensor
      LD      M10  ; .
      ANI     L10  ; Entry buffer pause mem
      AND     M133  ; Entry motor start mem
      ORB
      OUT     Y213  ; Entry motor
701   LD      M165  ; Front buffer motor start mem
      ANI     L11  ; Purify in buffer pause mem
      ANI     L12  ; Purify out buffer pause mem
      OUT     Y214  ; Buffer motor CR
705   LD      M123  ; #1-1Heating oven start mem
      OR      Y215  ; #1-1Heating oven air circulator
      ANI     T30  ; #1 Air circulator stop delay
      OUT     Y215  ; #1-1Heating oven air circulator
      ANI     M123  ; #1-1Heating oven start mem
      OUT     T30 K3000  ; #1 Air circulator stop delay
714   LD      M161  ; #1-2Heating oven start mem
      OR      Y216  ; #1-2Heating oven air circulator
      ANI     T32  ; #1-2 Air circulator stop delay
      OUT     Y216  ; #1-2Heating oven air circulator
      ANI     M161  ; #1-2Heating oven start mem
      OUT     T32 K3000  ; #1-2 Air circulator stop delay
723   LD      M102  ; Main start
      OR      L1  ; Water dropping force PB
      OUT     Y20E  ; Water drpping blower CR
726   LD      M102  ; Main start
      RST     L1  ; Water dropping force PB
728   LD      M131  ; De-reel start mem
      OUT     Y20F  ; De-reel motor CR
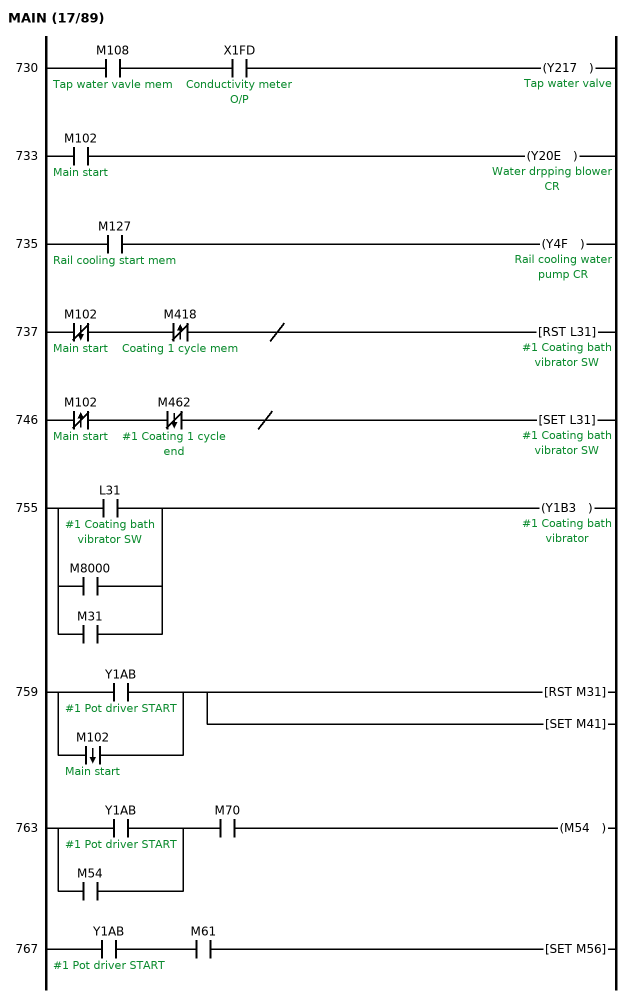
730   LD      M108  ; Tap water vavle mem
      AND     X1FD  ; Conductivity meter O/P
      OUT     Y217  ; Tap water valve
733   LD      M102  ; Main start
      OUT     Y20E  ; Water drpping blower CR
735   LD      M127  ; Rail cooling start mem
      OUT     Y4F  ; Rail cooling water pump CR
737   LDFI    M102  ; Main start
      ANDPI   M418  ; Coating 1 cycle mem
      INV
      RST     L31  ; #1 Coating bath vibrator SW
746   LDPI    M102  ; Main start
      ANDFI   M462  ; #1 Coating 1 cycle end
      INV
      SET     L31  ; #1 Coating bath vibrator SW
755   LD      L31  ; #1 Coating bath vibrator SW
      OR      M8000
      OR      M31
      OUT     Y1B3  ; #1 Coating bath vibrator
759   LD      Y1AB  ; #1 Pot driver START
      ORF     M102  ; Main start
      RST     M31
      SET     M41
763   LD      Y1AB  ; #1 Pot driver START
      OR      M54
      AND     M70
      OUT     M54
767   LD      Y1AB  ; #1 Pot driver START
      AND     M61
      SET     M56
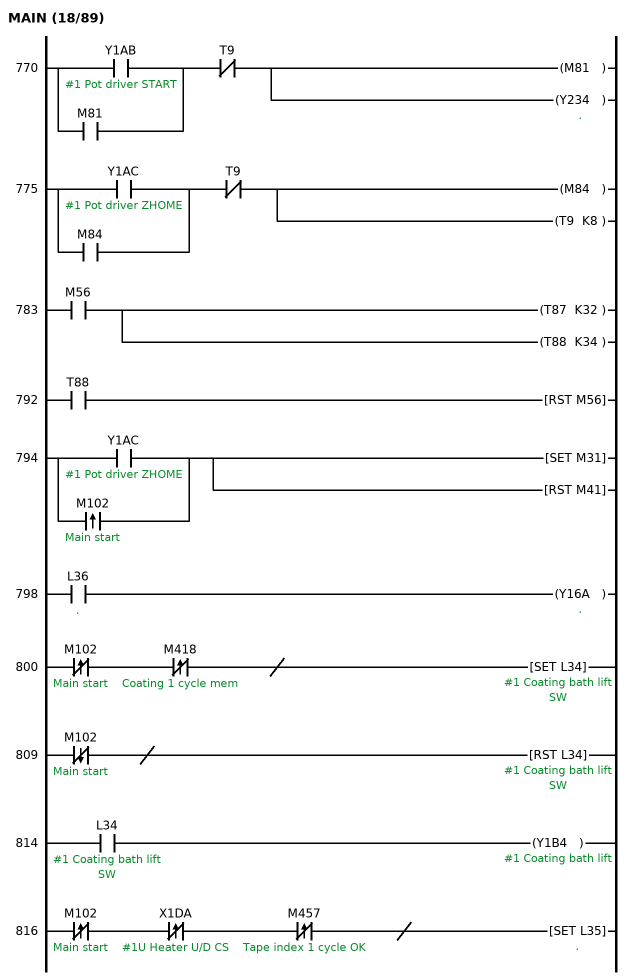
770   LD      Y1AB  ; #1 Pot driver START
      OR      M81
      ANI     T9
      OUT     M81
      OUT     Y234  ; .
775   LD      Y1AC  ; #1 Pot driver ZHOME
      OR      M84
      ANI     T9
      OUT     M84
      OUT     T9 K8
783   LD      M56
      OUT     T87 K32
      OUT     T88 K34
792   LD      T88
      RST     M56
794   LD      Y1AC  ; #1 Pot driver ZHOME
      ORP     M102  ; Main start
      SET     M31
      RST     M41
798   LD      L36  ; .
      OUT     Y16A  ; .
800   LDPI    M102  ; Main start
      ANDPI   M418  ; Coating 1 cycle mem
      INV
      SET     L34  ; #1 Coating bath lift SW
809   LDFI    M102  ; Main start
      INV
      RST     L34  ; #1 Coating bath lift SW
814   LD      L34  ; #1 Coating bath lift SW
      OUT     Y1B4  ; #1 Coating bath lift
816   LDPI    M102  ; Main start
      ANDPI   X1DA  ; #1U Heater U/D CS
      ANDPI   M457  ; Tape index 1 cycle OK
      INV
      SET     L35  ; .
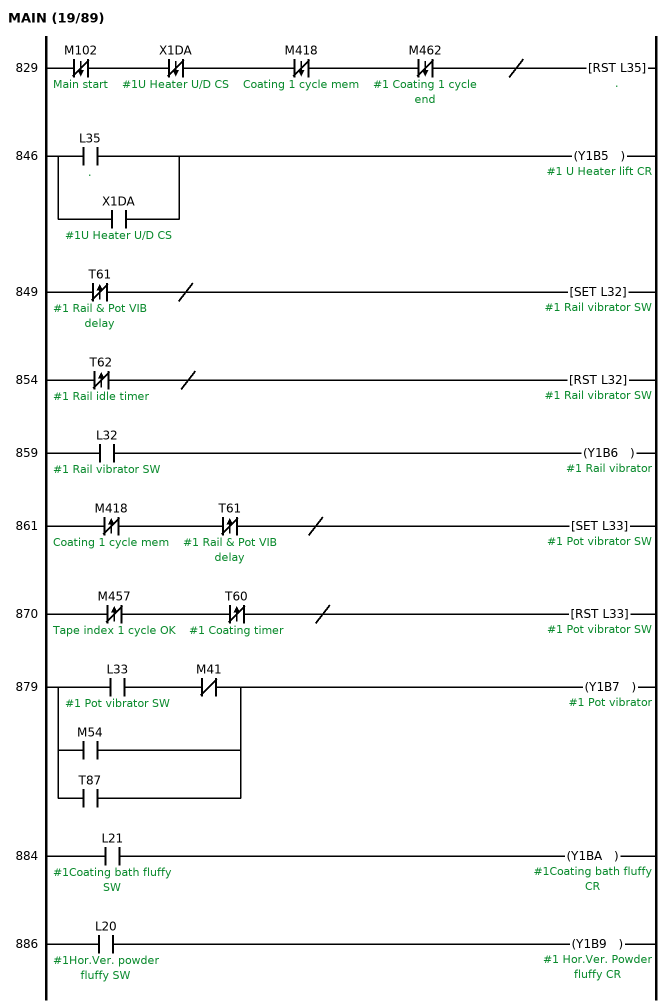
829   LDFI    M102  ; Main start
      ANDFI   X1DA  ; #1U Heater U/D CS
      ANDFI   M418  ; Coating 1 cycle mem
      ANDFI   M462  ; #1 Coating 1 cycle end
      INV
      RST     L35  ; .
846   LD      L35  ; .
      OR      X1DA  ; #1U Heater U/D CS
      OUT     Y1B5  ; #1 U Heater lift CR
849   LDPI    T61  ; #1 Rail & Pot VIB delay
      INV
      SET     L32  ; #1 Rail vibrator SW
854   LDPI    T62  ; #1 Rail idle timer
      INV
      RST     L32  ; #1 Rail vibrator SW
859   LD      L32  ; #1 Rail vibrator SW
      OUT     Y1B6  ; #1 Rail vibrator
861   LDPI    M418  ; Coating 1 cycle mem
      ANDPI   T61  ; #1 Rail & Pot VIB delay
      INV
      SET     L33  ; #1 Pot vibrator SW
870   LDPI    M457  ; Tape index 1 cycle OK
      ANDPI   T60  ; #1 Coating timer
      INV
      RST     L33  ; #1 Pot vibrator SW
879   LD      L33  ; #1 Pot vibrator SW
      ANI     M41
      OR      M54
      OR      T87
      OUT     Y1B7  ; #1 Pot vibrator
884   LD      L21  ; #1Coating bath fluffy SW
      OUT     Y1BA  ; #1Coating bath fluffy CR
886   LD      L20  ; #1Hor.Ver. powder fluffy SW
      OUT     Y1B9  ; #1 Hor.Ver. Powder fluffy CR
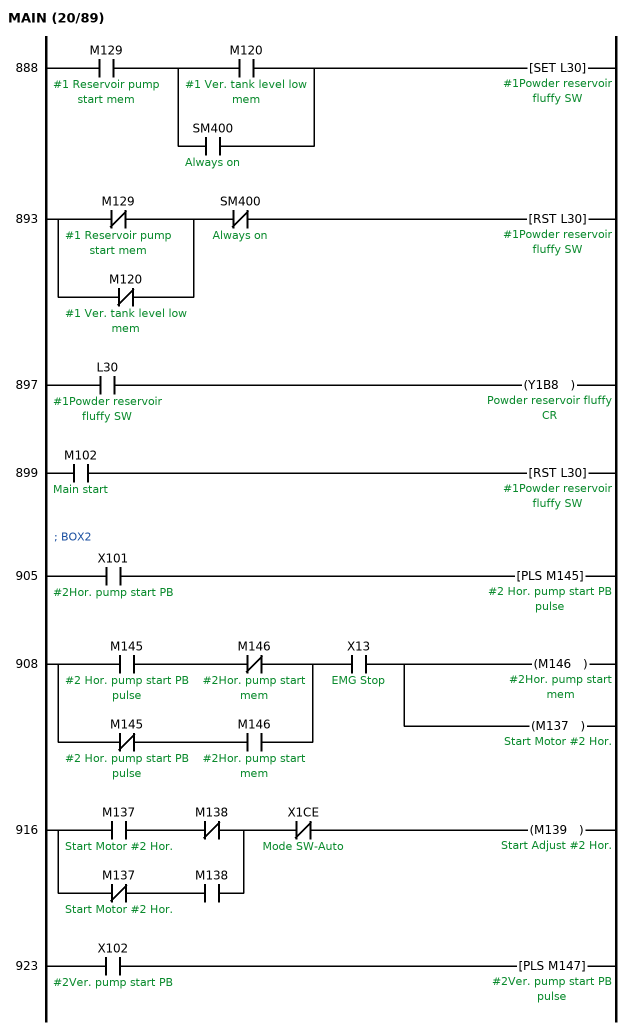
888   LD      M129  ; #1 Reservoir pump start mem
      LD      M120  ; #1 Ver. tank level low mem
      OR      SM400  ; Always on
      ANB
      SET     L30  ; #1Powder reservoir fluffy SW
893   LDI     M129  ; #1 Reservoir pump start mem
      ORI     M120  ; #1 Ver. tank level low mem
      ANI     SM400  ; Always on
      RST     L30  ; #1Powder reservoir fluffy SW
897   LD      L30  ; #1Powder reservoir fluffy SW
      OUT     Y1B8  ; Powder reservoir fluffy CR
899   LD      M102  ; Main start
      RST     L30  ; #1Powder reservoir fluffy SW
; BOX2
905   LD      X101  ; #2Hor. pump start PB
      PLS     M145  ; #2 Hor. pump start PB pulse
908   LD      M145  ; #2 Hor. pump start PB pulse
      ANI     M146  ; #2Hor. pump start mem
      LDI     M145  ; #2 Hor. pump start PB pulse
      AND     M146  ; #2Hor. pump start mem
      ORB
      AND     X13  ; EMG Stop
      OUT     M146  ; #2Hor. pump start mem
      OUT     M137  ; Start Motor #2 Hor.
916   LD      M137  ; Start Motor #2 Hor.
      ANI     M138
      LDI     M137  ; Start Motor #2 Hor.
      AND     M138
      ORB
      ANI     X1CE  ; Mode SW-Auto
      OUT     M139  ; Start Adjust #2 Hor.
923   LD      X102  ; #2Ver. pump start PB
      PLS     M147  ; #2Ver. pump start PB pulse
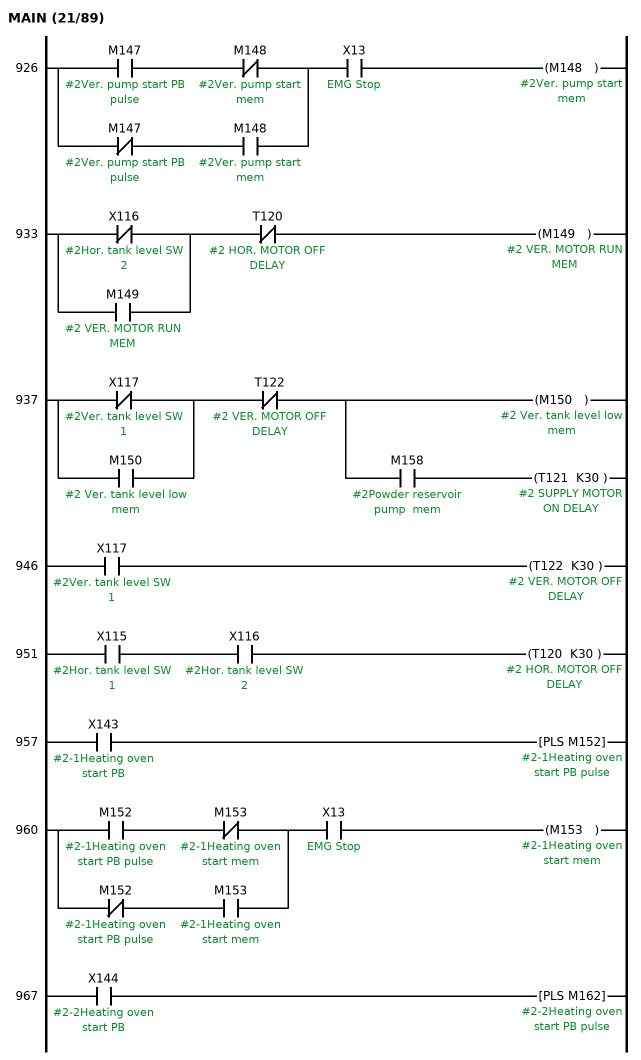
926   LD      M147  ; #2Ver. pump start PB pulse
      ANI     M148  ; #2Ver. pump start mem
      LDI     M147  ; #2Ver. pump start PB pulse
      AND     M148  ; #2Ver. pump start mem
      ORB
      AND     X13  ; EMG Stop
      OUT     M148  ; #2Ver. pump start mem
933   LDI     X116  ; #2Hor. tank level SW 2
      OR      M149  ; #2 VER. MOTOR RUN MEM
      ANI     T120  ; #2 HOR. MOTOR OFF DELAY
      OUT     M149  ; #2 VER. MOTOR RUN MEM
937   LDI     X117  ; #2Ver. tank level SW 1
      OR      M150  ; #2 Ver. tank level low mem
      ANI     T122  ; #2 VER. MOTOR OFF DELAY
      OUT     M150  ; #2 Ver. tank level low mem
      AND     M158  ; #2Powder reservoir pump  mem
      OUT     T121 K30  ; #2 SUPPLY MOTOR ON DELAY
946   LD      X117  ; #2Ver. tank level SW 1
      OUT     T122 K30  ; #2 VER. MOTOR OFF DELAY
951   LD      X115  ; #2Hor. tank level SW 1
      AND     X116  ; #2Hor. tank level SW 2
      OUT     T120 K30  ; #2 HOR. MOTOR OFF DELAY
957   LD      X143  ; #2-1Heating oven start PB
      PLS     M152  ; #2-1Heating oven start PB pulse
960   LD      M152  ; #2-1Heating oven start PB pulse
      ANI     M153  ; #2-1Heating oven start mem
      LDI     M152  ; #2-1Heating oven start PB pulse
      AND     M153  ; #2-1Heating oven start mem
      ORB
      AND     X13  ; EMG Stop
      OUT     M153  ; #2-1Heating oven start mem
967   LD      X144  ; #2-2Heating oven start PB
      PLS     M162  ; #2-2Heating oven start PB pulse
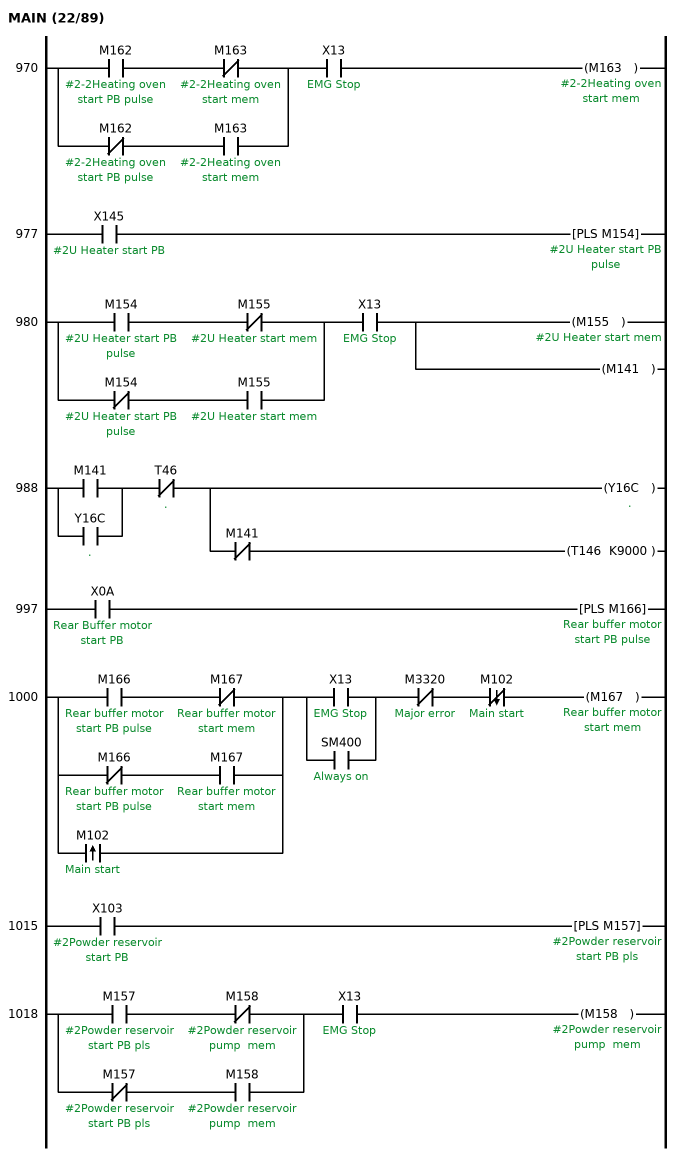
970   LD      M162  ; #2-2Heating oven start PB pulse
      ANI     M163  ; #2-2Heating oven start mem
      LDI     M162  ; #2-2Heating oven start PB pulse
      AND     M163  ; #2-2Heating oven start mem
      ORB
      AND     X13  ; EMG Stop
      OUT     M163  ; #2-2Heating oven start mem
977   LD      X145  ; #2U Heater start PB
      PLS     M154  ; #2U Heater start PB pulse
980   LD      M154  ; #2U Heater start PB pulse
      ANI     M155  ; #2U Heater start mem
      LDI     M154  ; #2U Heater start PB pulse
      AND     M155  ; #2U Heater start mem
      ORB
      AND     X13  ; EMG Stop
      OUT     M155  ; #2U Heater start mem
      OUT     M141
988   LD      M141
      OR      Y16C  ; .
      ANI     T46  ; .
      OUT     Y16C  ; .
      ANI     M141
      OUT     T146 K9000
997   LD      X0A  ; Rear Buffer motor start PB
      PLS     M166  ; Rear buffer motor start PB pulse
1000  LD      M166  ; Rear buffer motor start PB pulse
      ANI     M167  ; Rear buffer motor start mem
      LDI     M166  ; Rear buffer motor start PB pulse
      AND     M167  ; Rear buffer motor start mem
      ORB
      ORP     M102  ; Main start
      LD      X13  ; EMG Stop
      OR      SM400  ; Always on
      ANB
      ANI     M3320  ; Major error
      ANDFI   M102  ; Main start
      OUT     M167  ; Rear buffer motor start mem
1015  LD      X103  ; #2Powder reservoir start PB
      PLS     M157  ; #2Powder reservoir start PB pls
1018  LD      M157  ; #2Powder reservoir start PB pls
      ANI     M158  ; #2Powder reservoir pump  mem
      LDI     M157  ; #2Powder reservoir start PB pls
      AND     M158  ; #2Powder reservoir pump  mem
      ORB
      AND     X13  ; EMG Stop
      OUT     M158  ; #2Powder reservoir pump  mem
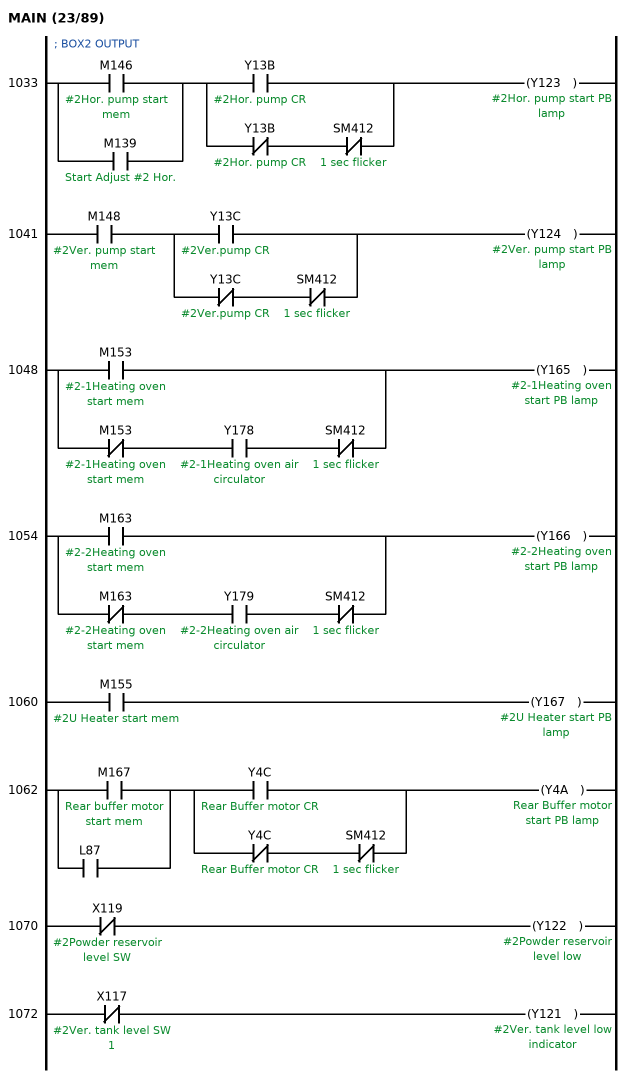
; BOX2 OUTPUT
1033  LD      M146  ; #2Hor. pump start mem
      OR      M139  ; Start Adjust #2 Hor.
      LD      Y13B  ; #2Hor. pump CR
      LDI     Y13B  ; #2Hor. pump CR
      ANI     SM412  ; 1 sec flicker
      ORB
      ANB
      OUT     Y123  ; #2Hor. pump start PB lamp
1041  LD      M148  ; #2Ver. pump start mem
      LD      Y13C  ; #2Ver.pump CR
      LDI     Y13C  ; #2Ver.pump CR
      ANI     SM412  ; 1 sec flicker
      ORB
      ANB
      OUT     Y124  ; #2Ver. pump start PB lamp
1048  LD      M153  ; #2-1Heating oven start mem
      LDI     M153  ; #2-1Heating oven start mem
      AND     Y178  ; #2-1Heating oven air circulator
      ANI     SM412  ; 1 sec flicker
      ORB
      OUT     Y165  ; #2-1Heating oven start PB lamp
1054  LD      M163  ; #2-2Heating oven start mem
      LDI     M163  ; #2-2Heating oven start mem
      AND     Y179  ; #2-2Heating oven air circulator
      ANI     SM412  ; 1 sec flicker
      ORB
      OUT     Y166  ; #2-2Heating oven start PB lamp
1060  LD      M155  ; #2U Heater start mem
      OUT     Y167  ; #2U Heater start PB lamp
1062  LD      M167  ; Rear buffer motor start mem
      OR      L87
      LD      Y4C  ; Rear Buffer motor CR
      LDI     Y4C  ; Rear Buffer motor CR
      ANI     SM412  ; 1 sec flicker
      ORB
      ANB
      OUT     Y4A  ; Rear Buffer motor start PB lamp
1070  LDI     X119  ; #2Powder reservoir level SW
      OUT     Y122  ; #2Powder reservoir level low
1072  LDI     X117  ; #2Ver. tank level SW 1
      OUT     Y121  ; #2Ver. tank level low indicator
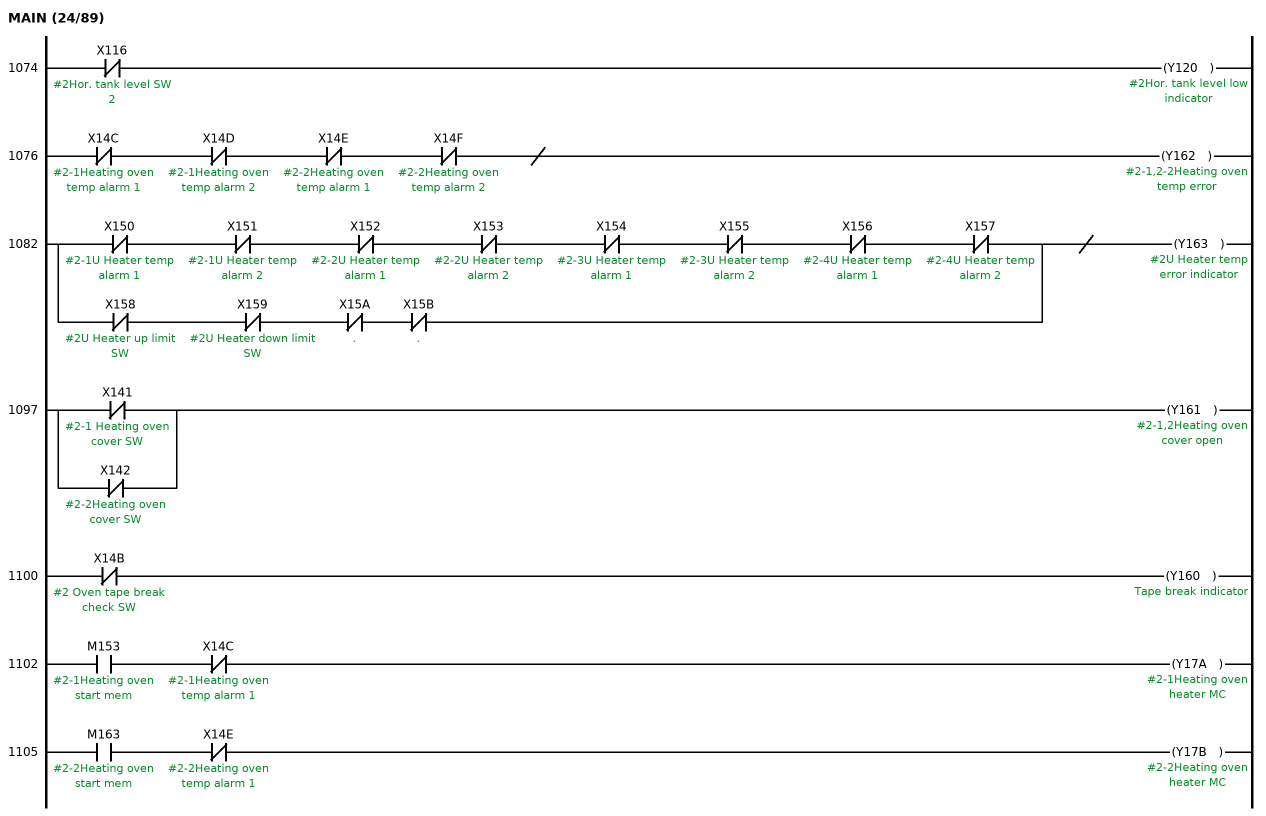
1074  LDI     X116  ; #2Hor. tank level SW 2
      OUT     Y120  ; #2Hor. tank level low indicator
1076  LDI     X14C  ; #2-1Heating oven temp alarm 1
      ANI     X14D  ; #2-1Heating oven temp alarm 2
      ANI     X14E  ; #2-2Heating oven temp alarm 1
      ANI     X14F  ; #2-2Heating oven temp alarm 2
      INV
      OUT     Y162  ; #2-1,2-2Heating oven temp error
1082  LDI     X150  ; #2-1U Heater temp alarm 1
      ANI     X151  ; #2-1U Heater temp alarm 2
      ANI     X152  ; #2-2U Heater temp alarm 1
      ANI     X153  ; #2-2U Heater temp alarm 2
      ANI     X154  ; #2-3U Heater temp alarm 1
      ANI     X155  ; #2-3U Heater temp alarm 2
      ANI     X156  ; #2-4U Heater temp alarm 1
      ANI     X157  ; #2-4U Heater temp alarm 2
      LDI     X158  ; #2U Heater up limit SW
      ANI     X159  ; #2U Heater down limit SW
      ANI     X15A  ; .
      ANI     X15B  ; .
      ORB
      INV
      OUT     Y163  ; #2U Heater temp error indicator
1097  LDI     X141  ; #2-1 Heating oven cover SW
      ORI     X142  ; #2-2Heating oven cover SW
      OUT     Y161  ; #2-1,2Heating oven cover open
1100  LDI     X14B  ; #2 Oven tape break check SW
      OUT     Y160  ; Tape break indicator
1102  LD      M153  ; #2-1Heating oven start mem
      ANI     X14C  ; #2-1Heating oven temp alarm 1
      OUT     Y17A  ; #2-1Heating oven heater MC
1105  LD      M163  ; #2-2Heating oven start mem
      ANI     X14E  ; #2-2Heating oven temp alarm 1
      OUT     Y17B  ; #2-2Heating oven heater MC
